///Datalogic output control
TYPE DatalogicOutputs :
STRUCT
    output1 : BIT; //Output 1
    output2 : BIT; //Output 2
    output3 : BIT; //Output 3
    ourput4 : BIT; //Output 4
    reserved1 : BIT;
    reserved2 : BIT;
    reserved3 : BIT;
    phaseTrigger : BIT; //Reading phase trigger
END_STRUCT
END_TYPE

(* stored: Version 1.1.0.1, ProductVersion 3.1.4020.12
   DUT DatalogicOutputs: Id {4ebf1db6-486f-429b-bcac-48af7d2b4f05} *)
